DATA_BLOCK "ST10_Stopper_InterfaceDB"
{ S7_Optimized_Access := 'TRUE' }
VERSION : 0.1
NON_RETAIN
   VAR
      aDev : Array[1..5] of "ST_Stopper";
      Command : Array[1..5] of "UDT_Stopper_FB";
   END_VAR


BEGIN

END_DATA_BLOCK

